Staubli VAL3: getOnline.pgx

public program getOnline(num handle_, bool& result_[])
begin
  // get mode of camera
  // result_ : true -> camera is online
  //         : false -> camera is offline
  call sendCommand(handle_,"go",result_)
end
